# B&R Automation Studio project MotionTestBenchMaster (part 16)

### HMI_PAM_1.typ
```iecst
(*HMI_PAM_1 Database for Filler PLC*)
(*Author = ????*)
(*DB Version : 0.10*)
(*File Version : 3.29*)

TYPE
        HMI_PAM_1_Type:     STRUCT
                            _000 : REAL; (*MOTORIZATION - Machine Slowing Speed [%]*)
                            _001 : REAL; (*MOTORIZATION - Machine Speed at Machine Empty [c/h]*)
                            _002 : REAL; (*MOTORIZATION - Machine Slowing Speed at End of Production [%]*)
                            _003 : REAL; (*MOTORIZATION - Machine Speed during Load/Unload Dummy Cans [c/h]*)
                            _004 : REAL; (*MOTORIZATION - Machine Speed on Cleaning/Sterilization [c/h]*)
                            _005 : REAL; (*MOTORIZATION - Machine Speed on External Cleaning and Washing [c/h]*)
                            _006 : REAL; (*MOTORIZATION - Machine Speed on Purge [c/h]*)
                            _007 : REAL; (*MOTORIZATION - Machine Speed on Caps Channel Emptying [c/h]*)
                            _008 : REAL; (*MOTORIZATION - Machine Speed on Rinse [c/h]*)
                            _009 : REAL; (*MOTORIZATION - Machine Speed during Containers Block [c/h]*)
                            _010 : REAL; (*MOTORIZATION - Motion JOG Speed [c/h]*)
                            _011 : REAL; (*MOTORIZATION - Motion Auto Acceleration  [s]*)
                            _012 : REAL; (*MOTORIZATION - Motion Auto Deceleration  [s]*)
                            _013 : REAL; (*MOTORIZATION - Motion Stop Position (0-XXX mm) [mm]*)
                            _014 : REAL; (*MOTORIZATION - Machine Speed on Rinser Control Insercion [c/h]*)
                            _015 : REAL; (*MOTORIZATION - Machine Speed on Rinser Control Continous [c/h]*)
                            _016 : REAL; (*MOTORIZATION - Spare *)
                            _017 : REAL; (*MOTORIZATION - Spare *)
                            _018 : REAL; (*MOTORIZATION - Spare *)
                            _019 : REAL; (*MOTORIZATION - Spare *)
                            _020 : REAL; (*MOTORIZATION - Machine Max Mechanical Speed [c/h]*)
                            _021 : REAL; (*MACHINE GREASING - Pause Laps Number *)
                            _022 : REAL; (*MACHINE GREASING - Greasing Cycles Number *)
                            _023 : REAL; (*MACHINE GREASING - Greasing Cycle Timeout [s]*)
                            _024 : REAL; (*SPARE - Spare *)
                            _025 : REAL; (*SPARE - Spare *)
                            _026 : REAL; (*SPARE - Spare *)
                            _027 : REAL; (*SPARE - Spare *)
                            _028 : REAL; (*SPARE - Spare *)
                            _029 : REAL; (*SPARE - Spare *)
                            _030 : REAL; (*COLLECTOR GREASING - Pause Laps Number *)
                            _031 : REAL; (*COLLECTOR GREASING - Greasing Cycles Number *)
                            _032 : REAL; (*COLLECTOR GREASING - Manual Cycles Number [s]*)
                            _033 : REAL; (*SPARE - Spare *)
                            _034 : REAL; (*SPARE - Spare *)
                            _035 : REAL; (*SPARE - Spare *)
                            _036 : REAL; (*FCI - First Containers Forced Rejected Enable *)
                            _037 : REAL; (*SPARE - Spare *)
                            _038 : REAL; (*SPARE - Spare *)
                            _039 : REAL; (*SPARE - Spare *)
                            _040 : REAL; (*OIL LUBRICATION - Pause Laps Number *)
                            _041 : REAL; (*OIL LUBRICATION - Working Laps Number *)
                            _042 : REAL; (*SPARE - Spare *)
                            _043 : REAL; (*SPARE - Spare *)
                            _044 : REAL; (*OIL LUBRICATION - Pause Laps Number *)
                            _045 : REAL; (*OIL LUBRICATION - Working Laps Number *)
                            _046 : REAL; (*WATER LUBRICATION - AVE260 - Pause Time With Bottles [s]*)
                            _047 : REAL; (*WATER LUBRICATION - AVE260 - Work Time With Bottles [s]*)
                            _048 : REAL; (*WATER LUBRICATION - Pause Laps Number *)
                            _049 : REAL; (*WATER LUBRICATION - Working Laps Number *)
                            _050 : REAL; (*WATER LUBRICATION - AVE260 - Pause Time Without Bottles [s]*)
                            _051 : REAL; (*WATER LUBRICATION - AVE260 - Work Time Without Bottles [s]*)
                            _052 : REAL; (*WATER LUBRICATION - AVE261 - Pause Time Without Bottles [s]*)
                            _053 : REAL; (*WATER LUBRICATION - AVE261 - Work Time Without Bottles [s]*)
                            _054 : REAL; (*WATER LUBRICATION - AVE261 - Enable Forced Time *)
                            _055 : REAL; (*WASHING - Cup Washing: Number of containers for washing during stop *)
                            _056 : REAL; (*WASHING - Cup Washing: Number of containers for forced washing *)
                            _057 : REAL; (*WATER LUBRICATION - AVE261 - Forced Pause Time Without Bottles *)
                            _058 : REAL; (*WATER LUBRICATION - AVE261 - Forced Work Time Without Bottles *)
                            _059 : REAL; (*SPARE - Spare *)
                            _060 : REAL; (*CONVEYOR - 257M1 - OUT Min [Hz]*)
                            _061 : REAL; (*CONVEYOR - 257M1 - OUT Max [Hz]*)
                            _062 : REAL; (*CONVEYOR - 257M1 - Spare [Hz]*)
                            _063 : REAL; (*CONVEYOR - 257M1 - Spare [Hz]*)
                            _064 : REAL; (*CONVEYOR - 257M1 - Spare [Hz]*)
                            _065 : REAL; (*CONVEYOR - Exit conveyor cleaning speed [Hz]*)
                            _066 : REAL; (*CONVEYOR - Spare *)
                            _067 : REAL; (*CONVEYOR - Spare *)
                            _068 : REAL; (*CONVEYOR - Spare *)
                            _069 : REAL; (*CONVEYOR - Spare *)
                            _070 : REAL; (*CONVEYOR - Spare *)
                            _071 : REAL; (*CONVEYOR - Spare *)
                            _072 : REAL; (*CONVEYOR - Spare *)
                            _073 : REAL; (*CONVEYOR - Spare *)
                            _074 : REAL; (*CONVEYOR - Spare *)
                            _075 : REAL; (*CONVEYOR - Spare *)
                            _076 : REAL; (*CONVEYOR - Spare *)
                            _077 : REAL; (*CONVEYOR - Spare *)
                            _078 : REAL; (*CONVEYOR - Spare *)
                            _079 : REAL; (*CONVEYOR - Spare *)
                            _080 : REAL; (*RINSER - Max Failed count Air Insercion control *)
                            _081 : REAL; (*RINSER - Max Failed count Water Insercion control *)
                            _082 : REAL; (*RINSER - Max Failed count Air Continous control *)
                            _083 : REAL; (*RINSER - Max Failed count Water Continus control *)
                            _084 : REAL; (*RINSER - Air Pressure threshold continous control [mbar]*)
                            _085 : REAL; (*RINSER - Water Pressure threshold continous control [mbar]*)
                            _086 : REAL; (*RINSER - Insercion Control Air Treatment Revolutions *)
                            _087 : REAL; (*RINSER - Insercion Control Water Treatment Revolutions *)
                            _088 : REAL; (*RINSER - Continous Control Air Treatment Revolutions *)
                            _089 : REAL; (*RINSER - Continous Control Water Treatment Revolutions *)
                            _090 : REAL; (*RINSER - Number of containers for forced insercion control *)
                            _091 : REAL; (*RINSER - Number of containers for forced continous control *)
                            _092 : REAL; (*RINSER - Rinser Water treatment pressure [bar]*)
                            _093 : REAL; (*RINSER - Rinser Cleaning solution pressure [bar]*)
                            _094 : REAL; (*SPARE - Spare *)
                            _095 : REAL; (*SPARE - Spare *)
                            _096 : REAL; (*SPARE - Spare *)
                            _097 : REAL; (*SPARE - Spare *)
                            _098 : REAL; (*SPARE - Spare *)
                            _099 : REAL; (*SPARE - Spare *)
                            _100 : REAL; (*BOTTOM COOLING - PPB205 Pump stroke [cm3/stroke]*)
                            _101 : REAL; (*BOTTOM COOLING - PPB205 Pure peracetic acid concentration [ppm]*)
                            _102 : REAL; (*BOTTOM COOLING - PPB205 Pure peracetic acid density [Kg/l]*)
                            _103 : REAL; (*BOTTOM COOLING - FTB205 Liter per pulse [l]*)
                            _104 : REAL; (*BOTTOM COOLING - Circuit capacity [l]*)
                            _105 : REAL; (*BOTTOM COOLING - PPB220 Delta on recipe set point for flow reduction [l/min]*)
                            _106 : REAL; (*BOTTOM COOLING - PPB220 Closed circuit flow set point [l/min]*)
                            _107 : REAL; (*BOTTOM COOLING - PPB220 Production Feed Forward [unit]*)
                            _108 : REAL; (*BOTTOM COOLING - Water temperature set point [°C]*)
                            _109 : REAL; (*BOTTOM COOLING - Delta on water temperature set point for alarm [°C]*)
                            _110 : REAL; (*BOTTOM COOLING - PPB220 high speed during CIP [Hz]*)
                            _111 : REAL; (*BOTTOM COOLING - PPB220 low speed during CIP [Hz]*)
                            _112 : REAL; (*BOTTOM COOLING - Collecting pipe filling time during CIP [s]*)
                            _113 : REAL; (*BOTTOM COOLING - Collecting pipe emptying time during CIP [s]*)
                            _114 : REAL; (*BOTTOM COOLING - Timeout UV Lamp water discharge at doors opening [min]*)
                            _115 : REAL; (*BOTTOM COOLING - Timeout UV Lamp water discharge during start up [s]*)
                            _116 : REAL; (*RINSER - PPB209 Low speed [Hz]*)
                            _117 : REAL; (*RINSER - PPB209 Medium speed [Hz]*)
                            _118 : REAL; (*RINSER - PPB209 High speed [Hz]*)
                            _119 : REAL; (*BOTTOM COOLING - Air temperature set point *)
                            _120 : REAL; (*BOTTOM COOLING - Delta on air temperature set point for alarm *)
                            _121 : REAL; (*SPARE - Spare *)
                            _122 : REAL; (*SPARE - Spare *)
                            _123 : REAL; (*SPARE - Spare *)
                            _124 : REAL; (*SPARE - Spare *)
                            _125 : REAL; (*SPARE - Spare *)
                            _126 : REAL; (*SPARE - Spare *)
                            _127 : REAL; (*SPARE - Spare *)
                            _128 : REAL; (*SPARE - Spare *)
                            _129 : REAL; (*SPARE - Spare *)
                            _130 : REAL; (*BOTTLE NECK WASHING - Set Point PID Temperature [°C]*)
                            _131 : REAL; (*BOTTLE NECK WASHING - Feed_Forward PID Temperature [%]*)
                            _132 : REAL; (*SPARE - Spare *)
                            _133 : REAL; (*SPARE - Spare *)
                            _134 : REAL; (*SPARE - Spare *)
                            _135 : REAL; (*SPARE - Spare *)
                            _136 : REAL; (*SPARE - Spare *)
                            _137 : REAL; (*SPARE - Spare *)
                            _138 : REAL; (*SPARE - Spare *)
                            _139 : REAL; (*SPARE - Spare *)
                            _140 : REAL; (*HYDRAULIC SEAL - PMI102 - Pump stroke [cm3/stroke]*)
                            _141 : REAL; (*HYDRAULIC SEAL - PMI102 - Pure peracetic acid concentration [ppm]*)
                            _142 : REAL; (*HYDRAULIC SEAL - PMI102 - Pure peracetic acid density [Kg/l]*)
                            _143 : REAL; (*HYDRAULIC SEAL - FTI101 - Liter per pulse [l]*)
                            _144 : REAL; (*HYDRAULIC SEAL - Circuit Capacity [l]*)
                            _145 : REAL; (*SPARE - Spare *)
                            _146 : REAL; (*SPARE - Spare *)
                            _147 : REAL; (*SPARE - Spare *)
                            _148 : REAL; (*SPARE - Spare *)
                            _149 : REAL; (*SPARE - Spare *)
                            _150 : REAL; (*STERILE WATER - PPW102 - Pump stroke [cm3/stroke]*)
                            _151 : REAL; (*STERILE WATER - PPW102 - Pure peracetic acid concentration [ppm]*)
                            _152 : REAL; (*STERILE WATER - PPW102 - Pure peracetic acid density [Kg/l]*)
                            _153 : REAL; (*STERILE WATER - PPW102 - Nitric acid concentration [ppm]*)
                            _154 : REAL; (*STERILE WATER - PPW102 - Nitric peracetic acid density [Kg/l]*)
                            _155 : REAL; (*STERILE WATER - PPW102 - Capacity for Purge Dosing Circuit [l]*)
                            _156 : REAL; (*STERILE WATER - PPW102 - Capacity for Purge Circuit [l]*)
                            _157 : REAL; (*SPARE - Spare *)
                            _158 : REAL; (*SPARE - Spare *)
                            _159 : REAL; (*SPARE - Spare *)
                            _160 : REAL; (*TREATMENT PREPARATION - CTP - Chemical (0: PAA 1: Clorine 2: Other) *)
                            _161 : REAL; (*TREATMENT PREPARATION - CTP - Pure chemical density [Kg/l]*)
                            _162 : REAL; (*TREATMENT PREPARATION - CTP - Flow meter position (0: Before 1:After) *)
                            _163 : REAL; (*TREATMENT PREPARATION - CTP - Dosing pump stroke [cm3/stroke]*)
                            _164 : REAL; (*TREATMENT PREPARATION - CTP - Chemical solution concentration [ppm]*)
                            _165 : REAL; (*TREATMENT PREPARATION - CTP - Inlet Water Flow Setpoint [l/min]*)
                            _166 : REAL; (*TREATMENT PREPARATION - CTP - Air Drying Pressure Setpoint [bar]*)
                            _167 : REAL; (*SPARE - Spare *)
                            _168 : REAL; (*SPARE - Spare *)
                            _169 : REAL; (*SPARE - Spare *)
                            _170 : REAL; (*WASHING - COP - Dosing Pump: Chemical (0: PAA 1: Clorine 2: Other) *)
                            _171 : REAL; (*WASHING - COP - Dosing Pump: Pure chemical density [Kg/l]*)
                            _172 : REAL; (*WASHING - COP - Dosing Pump: Flow meter position (0: Before 1:After) *)
                            _173 : REAL; (*WASHING - COP - Dosing Pump: Dosing pump stroke [cm3/stroke]*)
                            _174 : REAL; (*WASHING - COP - Dosing Pump: Chemical solution concentration [ppm]*)
                            _175 : REAL; (*WASHING - COP - Dosing Pump: Concentration Set Point [ppm]*)
                            _176 : REAL; (*SPARE - Spare *)
                            _177 : REAL; (*SPARE - Spare *)
                            _178 : REAL; (*SPARE - Spare *)
                            _179 : REAL; (*SPARE - Spare *)
                            _180 : REAL; (*WASHING - Enable Bottle Rejection after COP *)
                            _181 : REAL; (*WASHING - Number Of Bottles to Reject after COP *)
                            _182 : REAL; (*SPARE - Spare *)
                            _183 : REAL; (*SPARE - Spare *)
                            _184 : REAL; (*SPARE - Spare *)
                            _185 : REAL; (*SPARE - Spare *)
                            _186 : REAL; (*SPARE - Spare *)
                            _187 : REAL; (*SPARE - Spare *)
                            _188 : REAL; (*SPARE - Spare *)
                            _189 : REAL; (*SPARE - Spare *)
                            _190 : REAL; (*SPARE - Spare *)
                            _191 : REAL; (*SPARE - Spare *)
                            _192 : REAL; (*SPARE - Spare *)
                            _193 : REAL; (*SPARE - Spare *)
                            _194 : REAL; (*SPARE - Spare *)
                            _195 : REAL; (*SPARE - Spare *)
                            _196 : REAL; (*SPARE - Spare *)
                            _197 : REAL; (*SPARE - Spare *)
                            _198 : REAL; (*SPARE - Spare *)
                            _199 : REAL; (*SPARE - Spare *)
                            _200 : REAL; (*CAN SIZE - Conveyor Positioning Windows [mm]*)
                            _201 : REAL; (*CAN SIZE - Conveyor Gear IN *)
                            _202 : REAL; (*CAN SIZE - Conveyor Gear OUT *)
                            _203 : REAL; (*CAN SIZE - Conveyor Spindle Pitch *)
                            _204 : REAL; (*CAN SIZE - Conveyor Cleaning position [mm]*)
                            _205 : REAL; (*CAN SIZE - Spare *)
                            _206 : REAL; (*CAN SIZE - Spare *)
                            _207 : REAL; (*CAN SIZE - Spare *)
                            _208 : REAL; (*CAN SIZE - Spare *)
                            _209 : REAL; (*CAN SIZE - Spare *)
                            _210 : REAL; (*CAN SIZE - Spare *)
                            _211 : REAL; (*CAN SIZE - Spare *)
                            _212 : REAL; (*CAN SIZE - Spare *)
                            _213 : REAL; (*CAN SIZE - Spare *)
                            _214 : REAL; (*CAN SIZE - Spare *)
                            _215 : REAL; (*CAN SIZE - Conveyor Upper Limit [mm]*)
                            _216 : REAL; (*CAN SIZE - Conveyor Lower Limit [mm]*)
                            _217 : REAL; (*CAN SIZE - Conveyor Calibration Value *)
                            _218 : REAL; (*CAN SIZE - Conveyor Delta Inch *)
                            _219 : REAL; (*CAN SIZE - Spare *)
                            _220 : REAL; (*CAN SIZE - Guide Positioning Windows [mm]*)
                            _221 : REAL; (*CAN SIZE - Guide Gear IN *)
                            _222 : REAL; (*CAN SIZE - Guide Gear OUT *)
                            _223 : REAL; (*CAN SIZE - Guide Spindle Pitch *)
                            _224 : REAL; (*CAN SIZE - Guide Cleaning position [mm]*)
                            _225 : REAL; (*CAN SIZE - Spare *)
                            _226 : REAL; (*CAN SIZE - Spare *)
                            _227 : REAL; (*CAN SIZE - Spare *)
                            _228 : REAL; (*CAN SIZE - Spare *)
                            _229 : REAL; (*CAN SIZE - Spare *)
                            _230 : REAL; (*CAN SIZE - Spare *)
                            _231 : REAL; (*CAN SIZE - Spare *)
                            _232 : REAL; (*CAN SIZE - Spare *)
                            _233 : REAL; (*CAN SIZE - Spare *)
                            _234 : REAL; (*CAN SIZE - Spare *)
                            _235 : REAL; (*CAN SIZE - Guide Upper Limit [mm]*)
                            _236 : REAL; (*CAN SIZE - Guide Lower Limit [mm]*)
                            _237 : REAL; (*CAN SIZE - Guide Calibration Value *)
                            _238 : REAL; (*CAN SIZE - Guide Delta Inch *)
                            _239 : REAL; (*CAN SIZE - Spare *)
                            _240 : REAL; (*CAN SIZE - Spare *)
                            _241 : REAL; (*CAN SIZE - Spare *)
                            _242 : REAL; (*CAN SIZE - Spare *)
                            _243 : REAL; (*CAN SIZE - Spare *)
                            _244 : REAL; (*CAN SIZE - Spare *)
                            _245 : REAL; (*CAN SIZE - Spare *)
                            _246 : REAL; (*CAN SIZE - Spare *)
                            _247 : REAL; (*CAN SIZE - Spare *)
                            _248 : REAL; (*CAN SIZE - Spare *)
                            _249 : REAL; (*CAN SIZE - Spare *)
                            _250 : REAL; (*CAN SIZE - Tank position for Sampling  [mm]*)
                            _251 : REAL; (*CAN SIZE - Cam position for Sampling [mm]*)
                            _252 : REAL; (*CAN SIZE - Spare *)
                            _253 : REAL; (*CAN SIZE - Spare *)
                            _254 : REAL; (*CAN SIZE - Spare *)
                            _255 : REAL; (*CAN SIZE - Spare *)
                            _256 : REAL; (*CAN SIZE - Spare *)
                            _257 : REAL; (*CAN SIZE - Spare *)
                            _258 : REAL; (*CAN SIZE - Spare *)
                            _259 : REAL; (*CAN SIZE - Spare *)
                            _260 : REAL; (*CAN SIZE - Capper Size Change Motor 1 Low pos limit *)
                            _261 : REAL; (*CAN SIZE - Capper Size Change Motor 1 High pos limit *)
                            _262 : REAL; (*CAN SIZE - Capper Size Change Motor 2 Low pos limit *)
                            _263 : REAL; (*CAN SIZE - Capper Size Change Motor 2 High pos limit *)
                            _264 : REAL; (*CAN SIZE - Capper Size Change Motor 3 Low pos limit *)
                            _265 : REAL; (*CAN SIZE - Capper Size Change Motor 3 High pos limit *)
                            _266 : REAL; (*CAN SIZE - Capper Size Change Motor 1 Rotation direction *)
                            _267 : REAL; (*CAN SIZE - Capper Size Change Motor 2 Rotation direction *)
                            _268 : REAL; (*CAN SIZE - Capper Size Change Motor 3 Rotation direction *)
                            _269 : REAL; (*CAN SIZE - Capper Size Change Motor 1 Current Limit [A]*)
                            _270 : REAL; (*CAN SIZE - Capper Size Change Motor 2 Current Limit [A]*)
                            _271 : REAL; (*CAN SIZE - Capper Size Change Motor 3 Current Limit [A]*)
                            _272 : REAL; (*CAN SIZE - Capper Size Change Motor 1 Positioning Speed [rpm]*)
                            _273 : REAL; (*CAN SIZE - Capper Size Change Motor 2 Positioning Speed [rpm]*)
                            _274 : REAL; (*CAN SIZE - Capper Size Change Motor 3 Positioning Speed [rpm]*)
                            _275 : REAL; (*CAN SIZE - Capper Size Change Motor 1 Jog Speed [rpm]*)
                            _276 : REAL; (*CAN SIZE - Capper Size Change Motor 2 Jog Speed [rpm]*)
                            _277 : REAL; (*CAN SIZE - Capper Size Change Motor 3 Jog Speed [rpm]*)
                            _278 : REAL; (*CAN SIZE - Spare *)
                            _279 : REAL; (*CAN SIZE - Spare *)
                            _280 : REAL; (*CAN SIZE - Spare *)
                            _281 : REAL; (*CAN SIZE - Spare *)
                            _282 : REAL; (*CAN SIZE - Spare *)
                            _283 : REAL; (*CAN SIZE - Spare *)
                            _284 : REAL; (*CAN SIZE - Spare *)
                            _285 : REAL; (*CAN SIZE - Spare *)
                            _286 : REAL; (*CAN SIZE - Spare *)
                            _287 : REAL; (*CAN SIZE - Spare *)
                            _288 : REAL; (*CAN SIZE - Spare *)
                            _289 : REAL; (*CAN SIZE - Spare *)
                            _290 : REAL; (*CAN SIZE - Spare *)
                            _291 : REAL; (*CAN SIZE - Spare *)
                            _292 : REAL; (*CAN SIZE - Spare *)
                            _293 : REAL; (*CAN SIZE - Spare *)
                            _294 : REAL; (*CAN SIZE - Spare *)
                            _295 : REAL; (*CAN SIZE - Spare *)
                            _296 : REAL; (*CAN SIZE - Spare *)
                            _297 : REAL; (*CAN SIZE - Spare *)
                            _298 : REAL; (*CAN SIZE - Spare *)
                            _299 : REAL; (*CAN SIZE - Spare *)
                            _300 : REAL; (*WHITE ROOM - Basement fans standby speed [%]*)
                            _301 : REAL; (*WHITE ROOM - Basement fans production speed [%]*)
                            _302 : REAL; (*WHITE ROOM - Basement fans over speed [%]*)
                            _303 : REAL; (*WHITE ROOM - Spare *)
                            _304 : REAL; (*WHITE ROOM - Spare *)
                            _305 : REAL; (*WHITE ROOM - Filler fans standby speed [%]*)
                            _306 : REAL; (*WHITE ROOM - Filler fans production speed [%]*)
                            _307 : REAL; (*WHITE ROOM - Filler fans over speed [%]*)
                            _308 : REAL; (*WHITE ROOM - Spare *)
                            _309 : REAL; (*WHITE ROOM - Spare *)
                            _310 : REAL; (*WHITE ROOM - Rinser fans standby speed [%]*)
                            _311 : REAL; (*WHITE ROOM - Rinser fans production speed [%]*)
                            _312 : REAL; (*WHITE ROOM - Rinser fans over speed [%]*)
                            _313 : REAL; (*WHITE ROOM - Spare *)
                            _314 : REAL; (*WHITE ROOM - Spare *)
                            _315 : REAL; (*WHITE ROOM - Transfer fans standby speed [%]*)
                            _316 : REAL; (*WHITE ROOM - Transfer fans production speed [%]*)
                            _317 : REAL; (*WHITE ROOM - Transfer fans over speed [%]*)
                            _318 : REAL; (*WHITE ROOM - Spare *)
                            _319 : REAL; (*WHITE ROOM - Spare *)
                            _320 : REAL; (*WHITE ROOM - Seamer fans standby speed [%]*)
                            _321 : REAL; (*WHITE ROOM - Seamer fans production speed [%]*)
                            _322 : REAL; (*WHITE ROOM - Seamer fans over speed [%]*)
                            _323 : REAL; (*SPARE - Spare *)
                            _324 : REAL; (*SPARE - Spare *)
                            _325 : REAL; (*SPARE - Spare *)
                            _326 : REAL; (*SPARE - Spare *)
                            _327 : REAL; (*SPARE - Spare *)
                            _328 : REAL; (*SPARE - Spare *)
                            _329 : REAL; (*SPARE - Spare *)
                            _330 : REAL; (*SPARE - Spare *)
                            _331 : REAL; (*SPARE - Spare *)
                            _332 : REAL; (*SPARE - Spare *)
                            _333 : REAL; (*SPARE - Spare *)
                            _334 : REAL; (*SPARE - Spare *)
                            _335 : REAL; (*SPARE - Spare *)
                            _336 : REAL; (*SPARE - Spare *)
                            _337 : REAL; (*SPARE - Spare *)
                            _338 : REAL; (*SPARE - Spare *)
                            _339 : REAL; (*SPARE - Spare *)
                            _340 : REAL; (*SPARE - Spare *)
                            _341 : REAL; (*SPARE - Spare *)
                            _342 : REAL; (*SPARE - Spare *)
                            _343 : REAL; (*SPARE - Spare *)
                            _344 : REAL; (*SPARE - Spare *)
                            _345 : REAL; (*SPARE - Spare *)
                            _346 : REAL; (*SPARE - Spare *)
                            _347 : REAL; (*SPARE - Spare *)
                            _348 : REAL; (*SPARE - Spare *)
                            _349 : REAL; (*SPARE - Spare *)
                            _350 : REAL; (*SPARE - Spare *)
                            _351 : REAL; (*SPARE - Spare *)
                            _352 : REAL; (*SPARE - Spare *)
                            _353 : REAL; (*SPARE - Spare *)
                            _354 : REAL; (*SPARE - Spare *)
                            _355 : REAL; (*SPARE - Spare *)
                            _356 : REAL; (*SPARE - Spare *)
                            _357 : REAL; (*SPARE - Spare *)
                            _358 : REAL; (*SPARE - Spare *)
                            _359 : REAL; (*SPARE - Spare *)
                            _360 : REAL; (*SPARE - Spare *)
                            _361 : REAL; (*SPARE - Spare *)
                            _362 : REAL; (*SPARE - Spare *)
                            _363 : REAL; (*SPARE - Spare *)
                            _364 : REAL; (*SPARE - Spare *)
                            _365 : REAL; (*SPARE - Spare *)
                            _366 : REAL; (*SPARE - Spare *)
                            _367 : REAL; (*SPARE - Spare *)
                            _368 : REAL; (*SPARE - Spare *)
                            _369 : REAL; (*SPARE - Spare *)
                            _370 : REAL; (*SPARE - Spare *)
                            _371 : REAL; (*SPARE - Spare *)
                            _372 : REAL; (*SPARE - Spare *)
                            _373 : REAL; (*SPARE - Spare *)
                            _374 : REAL; (*SPARE - Spare *)
                            _375 : REAL; (*SPARE - Spare *)
                            _376 : REAL; (*SPARE - Spare *)
                            _377 : REAL; (*SPARE - Spare *)
                            _378 : REAL; (*SPARE - Spare *)
                            _379 : REAL; (*SPARE - Spare *)
                            _380 : REAL; (*SPARE - Spare *)
                            _381 : REAL; (*SPARE - Spare *)
                            _382 : REAL; (*SPARE - Spare *)
                            _383 : REAL; (*SPARE - Spare *)
                            _384 : REAL; (*SPARE - Spare *)
                            _385 : REAL; (*SPARE - Spare *)
                            _386 : REAL; (*SPARE - Spare *)
                            _387 : REAL; (*SPARE - Spare *)
                            _388 : REAL; (*SPARE - Spare *)
                            _389 : REAL; (*SPARE - Spare *)
                            _390 : REAL; (*SPARE - Spare *)
                            _391 : REAL; (*SPARE - Spare *)
                            _392 : REAL; (*SPARE - Spare *)
                            _393 : REAL; (*SPARE - Spare *)
                            _394 : REAL; (*SPARE - Spare *)
                            _395 : REAL; (*SPARE - Spare *)
                            _396 : REAL; (*MOTORIZATION - Cam 1 On Position [°]*)
                            _397 : REAL; (*MOTORIZATION - Cam 1 Off Position [°]*)
                            _398 : REAL; (*MOTORIZATION - Cam 1 Advanced Time [ms]*)
                            _399 : REAL; (*MOTORIZATION - Cam 1 Pulse numbers *)
                            _400 : REAL; (*MOTORIZATION - Cam 2 On Position [°]*)
                            _401 : REAL; (*MOTORIZATION - Cam 2 Off Position [°]*)
                            _402 : REAL; (*MOTORIZATION - Cam 2 Advanced Time [ms]*)
                            _403 : REAL; (*MOTORIZATION - Cam 2 Pulse numbers *)
                            _404 : REAL; (*MOTORIZATION - Cam 3 On Position [°]*)
                            _405 : REAL; (*MOTORIZATION - Cam 3 Off Position [°]*)
                            _406 : REAL; (*MOTORIZATION - Cam 3 Advanced Time [ms]*)
                            _407 : REAL; (*MOTORIZATION - Cam 3 Pulse numbers *)
                            _408 : REAL; (*MOTORIZATION - Cam 4 On Position [°]*)
                            _409 : REAL; (*MOTORIZATION - Cam 4 Off Position [°]*)
                            _410 : REAL; (*MOTORIZATION - Cam 4 Advanced Time [ms]*)
                            _411 : REAL; (*MOTORIZATION - Cam 4 Pulse numbers *)
                            _412 : REAL; (*MOTORIZATION - Cam 5 On Position [°]*)
                            _413 : REAL; (*MOTORIZATION - Cam 5 Off Position [°]*)
                            _414 : REAL; (*MOTORIZATION - Cam 5 Advanced Time [ms]*)
                            _415 : REAL; (*MOTORIZATION - Cam 5 Pulse numbers *)
                            _416 : REAL; (*MOTORIZATION - Cam 6 On Position [°]*)
                            _417 : REAL; (*MOTORIZATION - Cam 6 Off Position [°]*)
                            _418 : REAL; (*MOTORIZATION - Cam 6 Advanced Time [ms]*)
                            _419 : REAL; (*MOTORIZATION - Cam 6 Pulse numbers *)
                            _420 : REAL; (*MOTORIZATION - Cam 7 On Position [°]*)
                            _421 : REAL; (*MOTORIZATION - Cam 7 Off Position [°]*)
                            _422 : REAL; (*MOTORIZATION - Cam 7 Advanced Time [ms]*)
                            _423 : REAL; (*MOTORIZATION - Cam 7 Pulse numbers *)
                            _424 : REAL; (*MOTORIZATION - Cam 8 On Position [°]*)
                            _425 : REAL; (*MOTORIZATION - Cam 8 Off Position [°]*)
                            _426 : REAL; (*MOTORIZATION - Cam 8 Advanced Time [ms]*)
                            _427 : REAL; (*MOTORIZATION - Cam 8 Pulse numbers *)
                            _428 : REAL; (*MOTORIZATION - Cam 9 On Position [°]*)
                            _429 : REAL; (*MOTORIZATION - Cam 9 Off Position [°]*)
                            _430 : REAL; (*MOTORIZATION - Cam 9 Advanced Time [ms]*)
                            _431 : REAL; (*MOTORIZATION - Cam 9 Pulse numbers *)
                            _432 : REAL; (*MOTORIZATION - Cam 10 On Position [°]*)
                            _433 : REAL; (*MOTORIZATION - Cam 10 Off Position [°]*)
                            _434 : REAL; (*MOTORIZATION - Cam 10 Advanced Time [ms]*)
                            _435 : REAL; (*MOTORIZATION - Cam 10 Pulse numbers *)
                            _436 : REAL; (*MOTORIZATION - Cam 11 On Position [°]*)
                            _437 : REAL; (*MOTORIZATION - Cam 11 Off Position [°]*)
                            _438 : REAL; (*MOTORIZATION - Cam 11 Advanced Time [ms]*)
                            _439 : REAL; (*MOTORIZATION - Cam 11 Pulse Number  *)
                            _440 : REAL; (*MOTORIZATION - Spare *)
                            _441 : REAL; (*MOTORIZATION - Spare *)
                            _442 : REAL; (*MOTORIZATION - Spare *)
                            _443 : REAL; (*MOTORIZATION - Spare *)
                            _444 : REAL; (*MOTORIZATION - Spare *)
                            _445 : REAL; (*MOTORIZATION - Spare *)
                            _446 : REAL; (*MOTORIZATION - Spare *)
                            _447 : REAL; (*MOTORIZATION - Spare *)
                            _448 : REAL; (*MOTORIZATION - Spare *)
                            _449 : REAL; (*MOTORIZATION - Spare *)
                            _450 : REAL; (*CAPPER - Buffer Depth Cap Type 1 *)
                            _451 : REAL; (*CAPPER - Buffer Depth Cap Type 2 *)
                            _452 : REAL; (*CAPPER - Buffer Depth Cap Type 3 *)
                            _453 : REAL; (*CAPPER - Buffer Depth Cap Type 4 *)
                            _454 : REAL; (*CAPPER - Buffer Depth Max Limit *)
                            _455 : REAL; (*MOTORIZATION - Spare *)
                            _456 : REAL; (*MOTORIZATION - Spare *)
                            _457 : REAL; (*MOTORIZATION - Spare *)
                            _458 : REAL; (*MOTORIZATION - Spare *)
                            _459 : REAL; (*MOTORIZATION - Spare *)
                            _460 : REAL; (*MOTORIZATION - Spare *)
                            _461 : REAL; (*MOTORIZATION - Spare *)
                            _462 : REAL; (*MOTORIZATION - Spare *)
                            _463 : REAL; (*MOTORIZATION - Spare *)
                            _464 : REAL; (*MOTORIZATION - Spare *)
                            _465 : REAL; (*MOTORIZATION - Spare *)
                            _466 : REAL; (*MOTORIZATION - Spare *)
                            _467 : REAL; (*MOTORIZATION - Spare *)
                            _468 : REAL; (*MOTORIZATION - Spare *)
                            _469 : REAL; (*MOTORIZATION - Spare *)
                            _470 : REAL; (*MOTORIZATION - Spare *)
                            _471 : REAL; (*MOTORIZATION - Spare *)
                            _472 : REAL; (*MOTORIZATION - Spare *)
                            _473 : REAL; (*MOTORIZATION - Spare *)
                            _474 : REAL; (*MOTORIZATION - Spare *)
                            _475 : REAL; (*MOTORIZATION - Spare *)
                            _476 : REAL; (*MOTORIZATION - Spare *)
                            _477 : REAL; (*MOTORIZATION - Spare *)
                            _478 : REAL; (*MOTORIZATION - Spare *)
                            _479 : REAL; (*MOTORIZATION - Spare *)
                            _480 : REAL; (*MOTORIZATION - Spare *)
                            _481 : REAL; (*MOTORIZATION - Spare *)
                            _482 : REAL; (*MOTORIZATION - Spare *)
                            _483 : REAL; (*MOTORIZATION - Spare *)
                            _484 : REAL; (*MOTORIZATION - Spare *)
                            _485 : REAL; (*MOTORIZATION - Spare *)
                            _486 : REAL; (*MOTORIZATION - Spare *)
                            _487 : REAL; (*MOTORIZATION - Spare *)
                            _488 : REAL; (*MOTORIZATION - Spare *)
                            _489 : REAL; (*MOTORIZATION - Spare *)
                            _490 : REAL; (*MOTORIZATION - Spare *)
                            _491 : REAL; (*MOTORIZATION - Spare *)
                            _492 : REAL; (*MOTORIZATION - Spare *)
                            _493 : REAL; (*MOTORIZATION - Spare *)
                            _494 : REAL; (*MOTORIZATION - Spare *)
                            _495 : REAL; (*MOTORIZATION - Spare *)
                            _496 : REAL; (*MOTORIZATION - Spare *)
                            _497 : REAL; (*MOTORIZATION - Spare *)
                            _498 : REAL; (*MOTORIZATION - Spare *)
                            _499 : REAL; (*MOTORIZATION - Spare *)
                            _500 : REAL; (*MACHINE - 204DSF - Consecutive error counter preset - Machine Stop *)
                            _501 : REAL; (*MACHINE - 204DSF - Repetitive error counter preset - Bottle Stop *)
                            _502 : REAL; (*MACHINE - 204DSF - Absolute error counter preset - Machine Stop *)
                            _503 : REAL; (*MACHINE - 204DSF - Absolute error counter preset - Bottle Stop *)
                            _504 : REAL; (*MACHINE - 202DSF - Consecutive error counter preset - Machine Stop *)
                            _505 : REAL; (*MACHINE - 202DSF - Repetitive error counter preset - Bottle Stop *)
                            _506 : REAL; (*MACHINE - 202DSF - Absolute error counter preset - Machine Stop *)
                            _507 : REAL; (*MACHINE - 202DSF - Absolute error counter preset - Bottle Stop *)
                            _508 : REAL; (*MACHINE - 203DSF - Consecutive error counter preset - Machine Stop *)
                            _509 : REAL; (*MACHINE - 203DSF - Repetitive error counter preset - Bottle Stop *)
                            _510 : REAL; (*MACHINE - 203DSF - Absolute error counter preset - Machine Stop *)
                            _511 : REAL; (*MACHINE - 203DSF - Absolute error counter preset - Bottle Stop *)
                            _512 : REAL; (*MACHINE - 207DSF - Consecutive error counter preset - Machine Stop *)
                            _513 : REAL; (*MACHINE - 207DSF - Repetitive error counter preset - Bottle Stop *)
                            _514 : REAL; (*MACHINE - 207DSF - Absolute error counter preset - Machine Stop *)
                            _515 : REAL; (*MACHINE - 207DSF - Absolute error counter preset - Bottle Stop *)
                            _516 : REAL; (*MACHINE - 208DSF - Consecutive error counter preset - Machine Stop *)
                            _517 : REAL; (*MACHINE - 208DSF - Repetitive error counter preset - Bottle Stop *)
                            _518 : REAL; (*MACHINE - 208DSF - Absolute error counter preset - Machine Stop *)
                            _519 : REAL; (*MACHINE - 208DSF - Absolute error counter preset - Bottle Stop *)
                            _520 : REAL; (*MACHINE - 214CPB - Consecutive error counter preset - Machine Stop *)
                            _521 : REAL; (*MACHINE - 214CPB - Absolute error counter preset - Bottle Stop *)
                            _522 : REAL; (*SPARE - Spare *)
                            _523 : REAL; (*SPARE - Spare *)
                            _524 : REAL; (*MACHINE - 204DSB - Consecutive error counter preset - Machine Stop *)
                            _525 : REAL; (*MACHINE - 204DSB - Repetitive error counter preset - Bottle Stop *)
                            _526 : REAL; (*MACHINE - 204DSB - Absolute error counter preset - Machine Stop *)
                            _527 : REAL; (*MACHINE - 204DSB - Absolute error counter preset - Bottle Stop *)
                            _528 : REAL; (*SPARE - Spare *)
                            _529 : REAL; (*SPARE - Spare *)
                            _530 : REAL; (*SPARE - Spare *)
                            _531 : REAL; (*SPARE - Spare *)
                            _532 : REAL; (*SPARE - Spare *)
                            _533 : REAL; (*SPARE - Spare *)
                            _534 : REAL; (*SPARE - Spare *)
                            _535 : REAL; (*SPARE - Spare *)
                            _536 : REAL; (*SPARE - Spare *)
                            _537 : REAL; (*SPARE - Spare *)
                            _538 : REAL; (*SPARE - Spare *)
                            _539 : REAL; (*SPARE - Spare *)
                            _540 : REAL; (*SPARE - Spare *)
                            _541 : REAL; (*SPARE - Spare *)
                            _542 : REAL; (*SPARE - Spare *)
                            _543 : REAL; (*SPARE - Spare *)
                            _544 : REAL; (*SPARE - Spare *)
                            _545 : REAL; (*SPARE - Spare *)
                            _546 : REAL; (*SPARE - Spare *)
                            _547 : REAL; (*SPARE - Spare *)
                            _548 : REAL; (*SPARE - Spare *)
                            _549 : REAL; (*SPARE - Spare *)
                            _550 : REAL; (*MACHINE - 205EVB - Consecutive errors counter ejected - Machine Stop *)
                            _551 : REAL; (*MACHINE - 205EVB - Absolute errors counter ejected - Containers Stop *)
                            _552 : REAL; (*SPARE - Spare *)
                            _553 : REAL; (*SPARE - Spare *)
                            _554 : REAL; (*SPARE - Spare *)
                            _555 : REAL; (*SPARE - Spare *)
                            _556 : REAL; (*SPARE - Spare *)
                            _557 : REAL; (*SPARE - Spare *)
                            _558 : REAL; (*SPARE - Spare *)
                            _559 : REAL; (*MACHINE - Crowns Enable for Preclosed Bottles *)
                            _560 : REAL; (*MACHINE - Preclosing Laps Number for Bottle Burst *)
                            _561 : REAL; (*MACHINE - Preclosing Valves Number for Bottle Burst *)
                            _562 : REAL; (*MACHINE - Washing Laps Number for Bottle Burst *)
                            _563 : REAL; (*MACHINE - Bottel Burst washing pressure setpoint [bar]*)
                            _564 : REAL; (*MACHINE - Bottle Burst washing Low limit pressure [bar]*)
                            _565 : REAL; (*MACHINE - Preclosing Valves Number 1° Lap for Bottle Burst *)
                            _566 : REAL; (*MACHINE - Preclosing Valves Number 2° Lap for Bottle Burst *)
                            _567 : REAL; (*MACHINE - Preclosing Valves Number 3° Lap for Bottle Burst *)
                            _568 : REAL; (*MACHINE - Preclosing Valves Number 4° Lap for Bottle Burst *)
                            _569 : REAL; (*MACHINE - Preclosing Valves Number 5° Lap for Bottle Burst *)
                            _570 : REAL; (*SPARE - Spare *)
                            _571 : REAL; (*SPARE - Spare *)
                            _572 : REAL; (*SPARE - Spare *)
                            _573 : REAL; (*SPARE - Spare *)
                            _574 : REAL; (*SPARE - Spare *)
                            _575 : REAL; (*SPARE - Spare *)
                            _576 : REAL; (*SPARE - Spare *)
                            _577 : REAL; (*SPARE - Spare *)
                            _578 : REAL; (*SPARE - Spare *)
                            _579 : REAL; (*SPARE - Spare *)
                            _580 : REAL; (*SPARE - Spare *)
                            _581 : REAL; (*SPARE - Spare *)
                            _582 : REAL; (*SPARE - Spare *)
                            _583 : REAL; (*SPARE - Spare *)
                            _584 : REAL; (*SPARE - Spare *)
                            _585 : REAL; (*SPARE - Spare *)
                            _586 : REAL; (*SPARE - Spare *)
                            _587 : REAL; (*SPARE - Spare *)
                            _588 : REAL; (*SPARE - Spare *)
                            _589 : REAL; (*SPARE - Spare *)
                            _590 : REAL; (*SPARE - Spare *)
                            _591 : REAL; (*SPARE - Spare *)
                            _592 : REAL; (*SPARE - Spare *)
                            _593 : REAL; (*SPARE - Spare *)
                            _594 : REAL; (*SPARE - Spare *)
                            _595 : REAL; (*SPARE - Spare *)
                            _596 : REAL; (*SPARE - Spare *)
                            _597 : REAL; (*SPARE - Spare *)
                            _598 : REAL; (*SPARE - Spare *)
                            _599 : REAL; (*SPARE - Spare *)
                            _600 : REAL; (*SPARE - Spare *)
                            _601 : REAL; (*SPARE - Spare *)
                            _602 : REAL; (*SPARE - Spare *)
                            _603 : REAL; (*SPARE - Spare *)
                            _604 : REAL; (*SPARE - Spare *)
                            _605 : REAL; (*SPARE - Spare *)
                            _606 : REAL; (*SPARE - Spare *)
                            _607 : REAL; (*SPARE - Spare *)
                            _608 : REAL; (*SPARE - Spare *)
                            _609 : REAL; (*SPARE - Spare *)
                            _610 : REAL; (*SPARE - Spare *)
                            _611 : REAL; (*SPARE - Spare *)
                            _612 : REAL; (*SPARE - Spare *)
                            _613 : REAL; (*SPARE - Spare *)
                            _614 : REAL; (*SPARE - Spare *)
                            _615 : REAL; (*SPARE - Spare *)
                            _616 : REAL; (*SPARE - Spare *)
                            _617 : REAL; (*SPARE - Spare *)
                            _618 : REAL; (*SPARE - Spare *)
                            _619 : REAL; (*SPARE - Spare *)
                            _620 : REAL; (*SPARE - Spare *)
                            _621 : REAL; (*SPARE - Spare *)
                            _622 : REAL; (*SPARE - Spare *)
                            _623 : REAL; (*SPARE - Spare *)
                            _624 : REAL; (*SPARE - Spare *)
                            _625 : REAL; (*SPARE - Spare *)
                            _626 : REAL; (*SPARE - Spare *)
                            _627 : REAL; (*SPARE - Spare *)
                            _628 : REAL; (*SPARE - Spare *)
                            _629 : REAL; (*SPARE - Spare *)
                            _630 : REAL; (*SPARE - Spare *)
                            _631 : REAL; (*SPARE - Spare *)
                            _632 : REAL; (*SPARE - Spare *)
                            _633 : REAL; (*SPARE - Spare *)
                            _634 : REAL; (*SPARE - Spare *)
                            _635 : REAL; (*SPARE - Spare *)
                            _636 : REAL; (*SPARE - Spare *)
                            _637 : REAL; (*SPARE - Spare *)
                            _638 : REAL; (*SPARE - Spare *)
                            _639 : REAL; (*SPARE - Spare *)
                            _640 : REAL; (*SPARE - Spare *)
                            _641 : REAL; (*SPARE - Spare *)
                            _642 : REAL; (*SPARE - Spare *)
                            _643 : REAL; (*SPARE - Spare *)
                            _644 : REAL; (*SPARE - Spare *)
                            _645 : REAL; (*SPARE - Spare *)
                            _646 : REAL; (*SPARE - Spare *)
                            _647 : REAL; (*SPARE - Spare *)
                            _648 : REAL; (*SPARE - Spare *)
                            _649 : REAL; (*SPARE - Spare *)
                            _650 : REAL; (*SPARE - Spare *)
                            _651 : REAL; (*SPARE - Spare *)
                            _652 : REAL; (*SPARE - Spare *)
                            _653 : REAL; (*SPARE - Spare *)
                            _654 : REAL; (*SPARE - Spare *)
                            _655 : REAL; (*SPARE - Spare *)
                            _656 : REAL; (*SPARE - Spare *)
                            _657 : REAL; (*SPARE - Spare *)
                            _658 : REAL; (*SPARE - Spare *)
                            _659 : REAL; (*SPARE - Spare *)
                            _660 : REAL; (*SPARE - Spare *)
                            _661 : REAL; (*SPARE - Spare *)
                            _662 : REAL; (*SPARE - Spare *)
                            _663 : REAL; (*SPARE - Spare *)
                            _664 : REAL; (*SPARE - Spare *)
                            _665 : REAL; (*SPARE - Spare *)
                            _666 : REAL; (*SPARE - Spare *)
                            _667 : REAL; (*SPARE - Spare *)
                            _668 : REAL; (*SPARE - Spare *)
                            _669 : REAL; (*SPARE - Spare *)
                            _670 : REAL; (*SPARE - Spare *)
                            _671 : REAL; (*SPARE - Spare *)
                            _672 : REAL; (*SPARE - Spare *)
                            _673 : REAL; (*SPARE - Spare *)
                            _674 : REAL; (*SPARE - Spare *)
                            _675 : REAL; (*SPARE - Spare *)
                            _676 : REAL; (*SPARE - Spare *)
                            _677 : REAL; (*SPARE - Spare *)
                            _678 : REAL; (*SPARE - Spare *)
                            _679 : REAL; (*SPARE - Spare *)
                            _680 : REAL; (*SPARE - Spare *)
                            _681 : REAL; (*SPARE - Spare *)
                            _682 : REAL; (*SPARE - Spare *)
                            _683 : REAL; (*SPARE - Spare *)
                            _684 : REAL; (*SPARE - Spare *)
                            _685 : REAL; (*SPARE - Spare *)
                            _686 : REAL; (*SPARE - Spare *)
                            _687 : REAL; (*SPARE - Spare *)
                            _688 : REAL; (*SPARE - Spare *)
                            _689 : REAL; (*SPARE - Spare *)
                            _690 : REAL; (*SPARE - Spare *)
                            _691 : REAL; (*SPARE - Spare *)
                            _692 : REAL; (*SPARE - Spare *)
                            _693 : REAL; (*SPARE - Spare *)
                            _694 : REAL; (*SPARE - Spare *)
                            _695 : REAL; (*SPARE - Spare *)
                            _696 : REAL; (*SPARE - Spare *)
                            _697 : REAL; (*SPARE - Spare *)
                            _698 : REAL; (*SPARE - Spare *)
                            _699 : REAL; (*SPARE - Spare *)
                            _700 : REAL; (*SPARE - Spare *)
                            _701 : REAL; (*SPARE - Spare *)
                            _702 : REAL; (*SPARE - Spare *)
                            _703 : REAL; (*SPARE - Spare *)
                            _704 : REAL; (*SPARE - Spare *)
                            _705 : REAL; (*SPARE - Spare *)
                            _706 : REAL; (*SPARE - Spare *)
                            _707 : REAL; (*SPARE - Spare *)
                            _708 : REAL; (*SPARE - Spare *)
                            _709 : REAL; (*SPARE - Spare *)
                            _710 : REAL; (*SPARE - Spare *)
                            _711 : REAL; (*SPARE - Spare *)
                            _712 : REAL; (*SPARE - Spare *)
                            _713 : REAL; (*SPARE - Spare *)
                            _714 : REAL; (*SPARE - Spare *)
                            _715 : REAL; (*SPARE - Spare *)
                            _716 : REAL; (*SPARE - Spare *)
                            _717 : REAL; (*SPARE - Spare *)
                            _718 : REAL; (*SPARE - Spare *)
                            _719 : REAL; (*SPARE - Spare *)
                            _720 : REAL; (*SPARE - Spare *)
                            _721 : REAL; (*SPARE - Spare *)
                            _722 : REAL; (*SPARE - Spare *)
                            _723 : REAL; (*SPARE - Spare *)
                            _724 : REAL; (*SPARE - Spare *)
                            _725 : REAL; (*SPARE - Spare *)
                            _726 : REAL; (*SPARE - Spare *)
                            _727 : REAL; (*SPARE - Spare *)
                            _728 : REAL; (*SPARE - Spare *)
                            _729 : REAL; (*SPARE - Spare *)
                            _730 : REAL; (*SPARE - Spare *)
                            _731 : REAL; (*SPARE - Spare *)
                            _732 : REAL; (*SPARE - Spare *)
                            _733 : REAL; (*SPARE - Spare *)
                            _734 : REAL; (*SPARE - Spare *)
                            _735 : REAL; (*SPARE - Spare *)
                            _736 : REAL; (*SPARE - Spare *)
                            _737 : REAL; (*SPARE - Spare *)
                            _738 : REAL; (*SPARE - Spare *)
                            _739 : REAL; (*SPARE - Spare *)
                            _740 : REAL; (*SPARE - Spare *)
                            _741 : REAL; (*SPARE - Spare *)
                            _742 : REAL; (*SPARE - Spare *)
                            _743 : REAL; (*SPARE - Spare *)
                            _744 : REAL; (*SPARE - Spare *)
                            _745 : REAL; (*SPARE - Spare *)
                            _746 : REAL; (*SPARE - Spare *)
                            _747 : REAL; (*SPARE - Spare *)
                            _748 : REAL; (*SPARE - Spare *)
                            _749 : REAL; (*SPARE - Spare *)
                            _750 : REAL; (*SPARE - Spare *)
                            _751 : REAL; (*SPARE - Spare *)
                            _752 : REAL; (*SPARE - Spare *)
                            _753 : REAL; (*SPARE - Spare *)
                            _754 : REAL; (*SPARE - Spare *)
                            _755 : REAL; (*SPARE - Spare *)
                            _756 : REAL; (*SPARE - Spare *)
                            _757 : REAL; (*SPARE - Spare *)
                            _758 : REAL; (*SPARE - Spare *)
                            _759 : REAL; (*SPARE - Spare *)
                            _760 : REAL; (*SPARE - Spare *)
                            _761 : REAL; (*SPARE - Spare *)
                            _762 : REAL; (*SPARE - Spare *)
                            _763 : REAL; (*SPARE - Spare *)
                            _764 : REAL; (*SPARE - Spare *)
                            _765 : REAL; (*SPARE - Spare *)
                            _766 : REAL; (*SPARE - Spare *)
                            _767 : REAL; (*SPARE - Spare *)
                            _768 : REAL; (*SPARE - Spare *)
                            _769 : REAL; (*SPARE - Spare *)
                            _770 : REAL; (*SPARE - Spare *)
                            _771 : REAL; (*SPARE - Spare *)
                            _772 : REAL; (*SPARE - Spare *)
                            _773 : REAL; (*SPARE - Spare *)
                            _774 : REAL; (*SPARE - Spare *)
                            _775 : REAL; (*SPARE - Spare *)
                            _776 : REAL; (*SPARE - Spare *)
                            _777 : REAL; (*SPARE - Spare *)
                            _778 : REAL; (*SPARE - Spare *)
                            _779 : REAL; (*SPARE - Spare *)
                            _780 : REAL; (*SPARE - Spare *)
                            _781 : REAL; (*SPARE - Spare *)
                            _782 : REAL; (*SPARE - Spare *)
                            _783 : REAL; (*SPARE - Spare *)
                            _784 : REAL; (*SPARE - Spare *)
                            _785 : REAL; (*SPARE - Spare *)
                            _786 : REAL; (*SPARE - Spare *)
                            _787 : REAL; (*SPARE - Spare *)
                            _788 : REAL; (*SPARE - Spare *)
                            _789 : REAL; (*SPARE - Spare *)
                            _790 : REAL; (*SPARE - Spare *)
                            _791 : REAL; (*SPARE - Spare *)
                            _792 : REAL; (*SPARE - Spare *)
                            _793 : REAL; (*SPARE - Spare *)
                            _794 : REAL; (*SPARE - Spare *)
                            _795 : REAL; (*SPARE - Spare *)
                            _796 : REAL; (*SPARE - Spare *)
                            _797 : REAL; (*SPARE - Spare *)
                            _798 : REAL; (*SPARE - Spare *)
                            _799 : REAL; (*SPARE - Spare *)
                            _800 : REAL; (*SPARE - Spare *)
                            _801 : REAL; (*SPARE - Spare *)
                            _802 : REAL; (*SPARE - Spare *)
                            _803 : REAL; (*SPARE - Spare *)
                            _804 : REAL; (*SPARE - Spare *)
                            _805 : REAL; (*SPARE - Spare *)
                            _806 : REAL; (*SPARE - Spare *)
                            _807 : REAL; (*SPARE - Spare *)
                            _808 : REAL; (*SPARE - Spare *)
                            _809 : REAL; (*SPARE - Spare *)
                            _810 : REAL; (*SPARE - Spare *)
                            _811 : REAL; (*SPARE - Spare *)
                            _812 : REAL; (*SPARE - Spare *)
                            _813 : REAL; (*SPARE - Spare *)
                            _814 : REAL; (*SPARE - Spare *)
                            _815 : REAL; (*SPARE - Spare *)
                            _816 : REAL; (*SPARE - Spare *)
                            _817 : REAL; (*SPARE - Spare *)
                            _818 : REAL; (*SPARE - Spare *)
                            _819 : REAL; (*SPARE - Spare *)
                            _820 : REAL; (*SPARE - Spare *)
                            _821 : REAL; (*SPARE - Spare *)
                            _822 : REAL; (*SPARE - Spare *)
                            _823 : REAL; (*SPARE - Spare *)
                            _824 : REAL; (*SPARE - Spare *)
                            _825 : REAL; (*SPARE - Spare *)
                            _826 : REAL; (*SPARE - Spare *)
                            _827 : REAL; (*SPARE - Spare *)
                            _828 : REAL; (*SPARE - Spare *)
                            _829 : REAL; (*SPARE - Spare *)
                            _830 : REAL; (*SPARE - Spare *)
                            _831 : REAL; (*SPARE - Spare *)
                            _832 : REAL; (*SPARE - Spare *)
                            _833 : REAL; (*SPARE - Spare *)
                            _834 : REAL; (*SPARE - Spare *)
                            _835 : REAL; (*SPARE - Spare *)
                            _836 : REAL; (*SPARE - Spare *)
                            _837 : REAL; (*SPARE - Spare *)
                            _838 : REAL; (*SPARE - Spare *)
                            _839 : REAL; (*SPARE - Spare *)
                            _840 : REAL; (*SPARE - Spare *)
                            _841 : REAL; (*SPARE - Spare *)
                            _842 : REAL; (*SPARE - Spare *)
                            _843 : REAL; (*SPARE - Spare *)
                            _844 : REAL; (*SPARE - Spare *)
                            _845 : REAL; (*SPARE - Spare *)
                            _846 : REAL; (*SPARE - Spare *)
                            _847 : REAL; (*SPARE - Spare *)
                            _848 : REAL; (*SPARE - Spare *)
                            _849 : REAL; (*SPARE - Spare *)
                            _850 : REAL; (*SPARE - Spare *)
                            _851 : REAL; (*SPARE - Spare *)
                            _852 : REAL; (*SPARE - Spare *)
                            _853 : REAL; (*SPARE - Spare *)
                            _854 : REAL; (*SPARE - Spare *)
                            _855 : REAL; (*SPARE - Spare *)
                            _856 : REAL; (*SPARE - Spare *)
                            _857 : REAL; (*SPARE - Spare *)
                            _858 : REAL; (*SPARE - Spare *)
                            _859 : REAL; (*SPARE - Spare *)
                            _860 : REAL; (*SPARE - Spare *)
                            _861 : REAL; (*SPARE - Spare *)
                            _862 : REAL; (*SPARE - Spare *)
                            _863 : REAL; (*SPARE - Spare *)
                            _864 : REAL; (*SPARE - Spare *)
                            _865 : REAL; (*SPARE - Spare *)
                            _866 : REAL; (*SPARE - Spare *)
                            _867 : REAL; (*SPARE - Spare *)
                            _868 : REAL; (*SPARE - Spare *)
                            _869 : REAL; (*SPARE - Spare *)
                            _870 : REAL; (*SPARE - Spare *)
                            _871 : REAL; (*SPARE - Spare *)
                            _872 : REAL; (*SPARE - Spare *)
                            _873 : REAL; (*SPARE - Spare *)
                            _874 : REAL; (*SPARE - Spare *)
                            _875 : REAL; (*SPARE - Spare *)
                            _876 : REAL; (*SPARE - Spare *)
                            _877 : REAL; (*SPARE - Spare *)
                            _878 : REAL; (*SPARE - Spare *)
                            _879 : REAL; (*SPARE - Spare *)
                            _880 : REAL; (*SPARE - Spare *)
                            _881 : REAL; (*SPARE - Spare *)
                            _882 : REAL; (*SPARE - Spare *)
                            _883 : REAL; (*SPARE - Spare *)
                            _884 : REAL; (*SPARE - Spare *)
                            _885 : REAL; (*SPARE - Spare *)
                            _886 : REAL; (*SPARE - Spare *)
                            _887 : REAL; (*SPARE - Spare *)
                            _888 : REAL; (*SPARE - Spare *)
                            _889 : REAL; (*SPARE - Spare *)
                            _890 : REAL; (*SPARE - Spare *)
                            _891 : REAL; (*SPARE - Spare *)
                            _892 : REAL; (*SPARE - Spare *)
                            _893 : REAL; (*SPARE - Spare *)
                            _894 : REAL; (*SPARE - Spare *)
                            _895 : REAL; (*SPARE - Spare *)
                            _896 : REAL; (*SPARE - Spare *)
                            _897 : REAL; (*SPARE - Spare *)
                            _898 : REAL; (*SPARE - Spare *)
                            _899 : REAL; (*SPARE - Spare *)
                            _900 : REAL; (*CONTAINER SIZE - Container Size Max Volume (used only in PLC) *)
                            _901 : REAL; (*SPARE - Spare *)
                            _902 : REAL; (*SPARE - Spare *)
                            _903 : REAL; (*SPARE - Spare *)
                            _904 : REAL; (*SPARE - Spare *)
                            _905 : REAL; (*SPARE - Spare *)
                            _906 : REAL; (*SPARE - Spare *)
                            _907 : REAL; (*SPARE - Spare *)
                            _908 : REAL; (*SPARE - Spare *)
                            _909 : REAL; (*SPARE - Spare *)
                            _910 : REAL; (*SPARE - Spare *)
                            _911 : REAL; (*SPARE - Spare *)
                            _912 : REAL; (*SPARE - Spare *)
                            _913 : REAL; (*SPARE - Spare *)
                            _914 : REAL; (*SPARE - Spare *)
                            _915 : REAL; (*SPARE - Spare *)
                            _916 : REAL; (*SPARE - Spare *)
                            _917 : REAL; (*SPARE - Spare *)
                            _918 : REAL; (*SPARE - Spare *)
                            _919 : REAL; (*SPARE - Spare *)
                            _920 : REAL; (*SPARE - Spare *)
                            _921 : REAL; (*SPARE - Spare *)
                            _922 : REAL; (*SPARE - Spare *)
                            _923 : REAL; (*SPARE - Spare *)
                            _924 : REAL; (*SPARE - Spare *)
                            _925 : REAL; (*SPARE - Spare *)
                            _926 : REAL; (*SPARE - Spare *)
                            _927 : REAL; (*SPARE - Spare *)
                            _928 : REAL; (*SPARE - Spare *)
                            _929 : REAL; (*SPARE - Spare *)
                            _930 : REAL; (*SPARE - Spare *)
                            _931 : REAL; (*SPARE - Spare *)
                            _932 : REAL; (*SPARE - Spare *)
                            _933 : REAL; (*SPARE - Spare *)
                            _934 : REAL; (*SPARE - Spare *)
                            _935 : REAL; (*SPARE - Spare *)
                            _936 : REAL; (*SPARE - Spare *)
                            _937 : REAL; (*SPARE - Spare *)
                            _938 : REAL; (*SPARE - Spare *)
                            _939 : REAL; (*SPARE - Spare *)
                            _940 : REAL; (*SPARE - Spare *)
                            _941 : REAL; (*SPARE - Spare *)
                            _942 : REAL; (*SPARE - Spare *)
                            _943 : REAL; (*SPARE - Spare *)
                            _944 : REAL; (*SPARE - Spare *)
                            _945 : REAL; (*SPARE - Spare *)
                            _946 : REAL; (*SPARE - Spare *)
                            _947 : REAL; (*SPARE - Spare *)
                            _948 : REAL; (*SPARE - Spare *)
                            _949 : REAL; (*SPARE - Spare *)
                            _950 : REAL; (*SPARE - Spare *)
                            _951 : REAL; (*SPARE - Spare *)
                            _952 : REAL; (*SPARE - Spare *)
                            _953 : REAL; (*SPARE - Spare *)
                            _954 : REAL; (*SPARE - Spare *)
                            _955 : REAL; (*SPARE - Spare *)
                            _956 : REAL; (*SPARE - Spare *)
                            _957 : REAL; (*SPARE - Spare *)
                            _958 : REAL; (*SPARE - Spare *)
                            _959 : REAL; (*SPARE - Spare *)
                            _960 : REAL; (*SPARE - Spare *)
                            _961 : REAL; (*SPARE - Spare *)
                            _962 : REAL; (*SPARE - Spare *)
                            _963 : REAL; (*SPARE - Spare *)
                            _964 : REAL; (*SPARE - Spare *)
                            _965 : REAL; (*SPARE - Spare *)
                            _966 : REAL; (*SPARE - Spare *)
                            _967 : REAL; (*SPARE - Spare *)
                            _968 : REAL; (*SPARE - Spare *)
                            _969 : REAL; (*SPARE - Spare *)
                            _970 : REAL; (*SPARE - Spare *)
                            _971 : REAL; (*SPARE - Spare *)
                            _972 : REAL; (*SPARE - Spare *)
                            _973 : REAL; (*SPARE - Spare *)
                            _974 : REAL; (*SPARE - Spare *)
                            _975 : REAL; (*SPARE - Spare *)
                            _976 : REAL; (*SPARE - Spare *)
                            _977 : REAL; (*SPARE - Spare *)
                            _978 : REAL; (*SPARE - Spare *)
                            _979 : REAL; (*SPARE - Spare *)
                            _980 : REAL; (*SPARE - Spare *)
                            _981 : REAL; (*SPARE - Spare *)
                            _982 : REAL; (*SPARE - Spare *)
                            _983 : REAL; (*SPARE - Spare *)
                            _984 : REAL; (*SPARE - Spare *)
                            _985 : REAL; (*SPARE - Spare *)
                            _986 : REAL; (*SPARE - Spare *)
                            _987 : REAL; (*SPARE - Spare *)
                            _988 : REAL; (*SPARE - Spare *)
                            _989 : REAL; (*SPARE - Spare *)
                            _990 : REAL; (*SPARE - Spare *)
                            _991 : REAL; (*SPARE - Spare *)
                            _992 : REAL; (*SPARE - Spare *)
                            _993 : REAL; (*SPARE - Spare *)
                            _994 : REAL; (*SPARE - Spare *)
                            _995 : REAL; (*SPARE - Spare *)
                            _996 : REAL; (*SPARE - Spare *)
                            _997 : REAL; (*SPARE - Spare *)
                            _998 : REAL; (*SPARE - Spare *)
                            _999 : REAL; (*SPARE - Spare *)
        END_STRUCT;
END_TYPE
```
